FUNCTION_BLOCK HaltedUnifiedProgramState EXTENDS HaltedProgramState
VAR
	{attribute 'OPC.UA.DA' := '0'}
	_ClassName : STRING := __POUNAME();
END_VAR

{attribute 'monitoring' := 'call'}
PROPERTY ClassName : STRING
GET
ClassName := _ClassName;
END_GET
END_PROPERTY

END_FUNCTION_BLOCK

(* stored: Version 1.1.0.1
   POU HaltedUnifiedProgramState: Id {89ef2886-2d89-45dd-b318-52671d3dd7ba}, SpecialFunc None
   Property ClassName: Id {e418ea27-4a57-4e13-a753-11485adbb071}
   Get Get: Id {38309879-9702-4b79-9478-100eff5864a1} *)
